PROGRAM X02_Database (*always run this FB in a 1ms task*)
VAR

	tonStartUpDelay		: TON;
	fbPulse_RepeatConnectionAttempt				: FB_PulseGenerator;

	fbDB_CreateConnection: FB_DB_CreateConnectionParams;
	(*fbAuxilaryPCV: FB_DB_PCV_Check;
	fbPCV: FB_DB_PCV_Check;
	fbOCV: FB_DB_OCV_Check;
	fbOAC: FB_DB_OAC_Check;
	fbCAC: FB_DB_CAC_Check;*)


	fbDBReport	: FB_DB_ReportExeSP;

	test : BOOL;

END_VAR

(*
Modification history:
Date		|	Author 		|	Remark
----------------------------------------------------------------------------------------------------
03.09.20	|	PP			|	Start Remarking.
*)

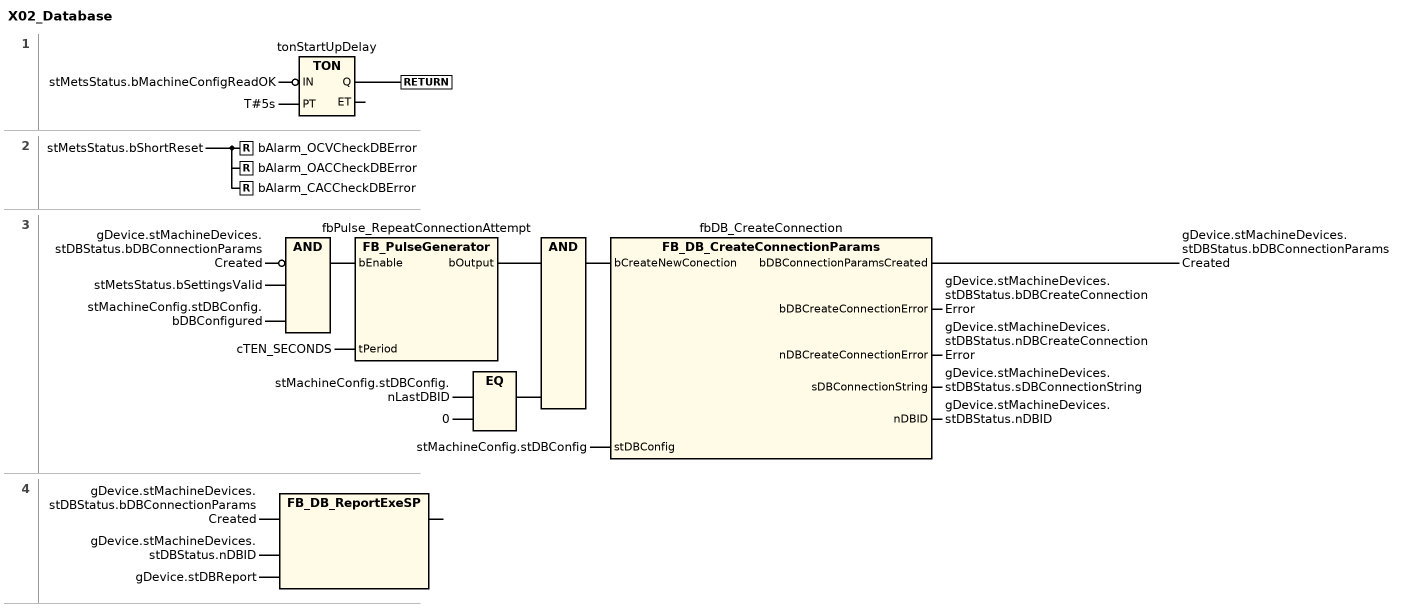
// NETWORK 1
tonStartUpDelay(IN := NOT stMetsStatus.bMachineConfigReadOK, PT := T#5s); // TON
IF tonStartUpDelay.Q THEN RETURN; END_IF

// NETWORK 2
bAlarm_OCVCheckDBError R= stMetsStatus.bShortReset;
bAlarm_OACCheckDBError R= stMetsStatus.bShortReset;
bAlarm_CACCheckDBError R= stMetsStatus.bShortReset;

// NETWORK 3
fbPulse_RepeatConnectionAttempt(bEnable := NOT gDevice.stMachineDevices.stDBStatus.bDBConnectionParamsCreated AND stMetsStatus.bSettingsValid AND stMachineConfig.stDBConfig.bDBConfigured, tPeriod := cTEN_SECONDS); // FB_PulseGenerator
fbDB_CreateConnection(
    bCreateNewConection := fbPulse_RepeatConnectionAttempt.bOutput AND stMachineConfig.stDBConfig.nLastDBID = 0,
    stDBConfig := stMachineConfig.stDBConfig,
    bDBCreateConnectionError => gDevice.stMachineDevices.stDBStatus.bDBCreateConnectionError,
    nDBCreateConnectionError => gDevice.stMachineDevices.stDBStatus.nDBCreateConnectionError,
    sDBConnectionString => gDevice.stMachineDevices.stDBStatus.sDBConnectionString,
    nDBID => gDevice.stMachineDevices.stDBStatus.nDBID); // FB_DB_CreateConnectionParams
gDevice.stMachineDevices.stDBStatus.bDBConnectionParamsCreated := fbDB_CreateConnection.bDBConnectionParamsCreated;

// NETWORK 4
FB_DB_ReportExeSP(gDevice.stMachineDevices.stDBStatus.bDBConnectionParamsCreated, gDevice.stMachineDevices.stDBStatus.nDBID, gDevice.stDBReport);

END_PROGRAM

(* stored: Version 1.1.0.1
   POU X02_Database: Id {dae25524-1c6e-4864-a24d-1db29e52ccea}, SpecialFunc None *)
